// TIA Portal V20 export
TYPE "LConSMC_typeActualDynamics"
// stored: Access Published
   STRUCT
      s : LReal;   // Position
      v : LReal;   // Speed
      "a" : LReal;   // Acceleration
      d : LReal;   // Deceleration
      j : LReal;   // Jerk
   END_STRUCT;
END_TYPE
